(* IEC 61131-3 sources: eCockpitGit/test_project/src/%F%00 Library/%F%Common Functions/%F%Bits/%F%Bit Set Part Through, 8 files *)

(* ---- %POU%FU_bBitPartThrough.st ---- *)
//This function changed only the needed bits of a variable
// |**Version**|**Author**| **Date** |**Changes**
// | 1         | NSN      | 16-03-22 | Creation
FUNCTION FU_bBitPartThrough : BYTE
VAR_INPUT
	valueChange		:BYTE;		//Variable to change
	value			:BYTE;		//Value to change bits to
	amount			:BYTE;		//Amount of bits to change
	offset			:BYTE;		//Offset in variable to change bits at
END_VAR
(*%!%__DELIMITER__%!%*)
FU_bBitPartThrough		:=		(valueChange AND ROL(GConstants.binaryInvMaskByte[amount],offset)) OR SHL(value AND GConstants.binaryMaskByte[amount],offset);

(* ---- %POU%FU_diBitPartThrough.st ---- *)
//This function changed only the needed bits of a variable
// |**Version**|**Author**| **Date** |**Changes**
// | 1         | NSN      | 16-03-22 | Creation
FUNCTION FU_diBitPartThrough : DINT
VAR_INPUT
	valueChange		:DINT;		//Variable to change
	value			:DINT;		//Value to change bits to
	amount			:BYTE;		//Amount of bits to change
	offset			:BYTE;		//Offset in variable to change bits at
END_VAR
(*%!%__DELIMITER__%!%*)
FU_diBitPartThrough		:=		TO_DINT((TO_DWORD(valueChange) AND ROL(GConstants.binaryInvMaskDWord[amount],offset)) OR SHL(TO_DWORD(value) AND GConstants.binaryMaskDWord[amount],offset));

(* ---- %POU%FU_dwBitPartThrough.st ---- *)
//This function changed only the needed bits of a variable
// |**Version**|**Author**| **Date** |**Changes**
// | 1         | NSN      | 16-03-22 | Creation
FUNCTION FU_dwBitPartThrough : DWORD
VAR_INPUT
	valueChange		:DWORD;		//Variable to change
	value			:DWORD;		//Value to change bits to
	amount			:BYTE;		//Amount of bits to change
	offset			:BYTE;		//Offset in variable to change bits at
END_VAR
(*%!%__DELIMITER__%!%*)
FU_dwBitPartThrough		:=		(valueChange AND ROL(GConstants.binaryInvMaskDWord[amount],offset)) OR SHL(value AND GConstants.binaryMaskDWord[amount],offset);

(* ---- %POU%FU_iBitPartThrough.st ---- *)
//This function changed only the needed bits of a variable
// |**Version**|**Author**| **Date** |**Changes**
// | 1         | NSN      | 16-03-22 | Creation
FUNCTION FU_iBitPartThrough : INT
VAR_INPUT
	valueChange		:INT;		//Variable to change
	value			:INT;		//Value to change bits to
	amount			:BYTE;		//Amount of bits to change
	offset			:BYTE;		//Offset in variable to change bits at
END_VAR
(*%!%__DELIMITER__%!%*)
FU_iBitPartThrough		:=		TO_INT((TO_UINT(valueChange) AND ROL(TO_UINT(GConstants.binaryInvMaskInt[amount]),offset)) OR SHL(TO_UINT(value) AND TO_UINT(GConstants.binaryMaskInt[amount]),offset));

(* ---- %POU%FU_liBitPartThrough.st ---- *)
//This function changed only the needed bits of a variable
// |**Version**|**Author**| **Date** |**Changes**
// | 1         | NSN      | 16-03-22 | Creation
FUNCTION FU_liBitPartThrough : LINT
VAR_INPUT
	valueChange		:LINT;		//Variable to change
	value			:LINT;		//Value to change bits to
	amount			:BYTE;		//Amount of bits to change
	offset			:BYTE;		//Offset in variable to change bits at
END_VAR
(*%!%__DELIMITER__%!%*)
FU_liBitPartThrough		:=		TO_LINT((TO_LWORD(valueChange) AND ROL(GConstants.binaryInvMaskLWord[amount],offset)) OR SHL(TO_LWORD(value) AND GConstants.binaryMaskLWord[amount],offset));

(* ---- %POU%FU_lwBitPartThrough.st ---- *)
//This function changed only the needed bits of a variable
// |**Version**|**Author**| **Date** |**Changes**
// | 1         | NSN      | 16-03-22 | Creation
FUNCTION FU_lwBitPartThrough : LWORD
VAR_INPUT
	valueChange		:LWORD;		//Variable to change
	value			:LWORD;		//Value to change bits to
	amount			:BYTE;		//Amount of bits to change
	offset			:BYTE;		//Offset in variable to change bits at
END_VAR
(*%!%__DELIMITER__%!%*)
FU_lwBitPartThrough		:=		(valueChange AND ROL(GConstants.binaryInvMaskLWord[amount],offset)) OR SHL(value AND GConstants.binaryMaskLWord[amount],offset);

(* ---- %POU%FU_siBitPartThrough.st ---- *)
//This function changed only the needed bits of a variable
// |**Version**|**Author**| **Date** |**Changes**
// | 1         | NSN      | 16-03-22 | Creation
FUNCTION FU_siBitPartThrough : SINT
VAR_INPUT
	valueChange		:SINT;		//Variable to change
	value			:SINT;		//Value to change bits to
	amount			:BYTE;		//Amount of bits to change
	offset			:BYTE;		//Offset in variable to change bits at
END_VAR
(*%!%__DELIMITER__%!%*)
FU_siBitPartThrough		:=		TO_SINT((TO_USINT(valueChange) AND ROL(TO_USINT(GConstants.binaryInvMaskSint[amount]),offset)) OR SHL(TO_USINT(value) AND TO_USINT(GConstants.binaryMaskSint[amount]),offset));

(* ---- %POU%FU_wBitPartThrough.st ---- *)
//This function changed only the needed bits of a variable
// |**Version**|**Author**| **Date** |**Changes**
// | 1         | NSN      | 16-03-22 | Creation
FUNCTION FU_wBitPartThrough : WORD
VAR_INPUT
	valueChange		:WORD;		//Variable to change
	value			:WORD;		//Value to change bits to
	amount			:BYTE;		//Amount of bits to change
	offset			:BYTE;		//Offset in variable to change bits at
END_VAR
(*%!%__DELIMITER__%!%*)
FU_wBitPartThrough		:=		(valueChange AND ROL(GConstants.binaryInvMaskWord[amount],offset)) OR SHL(value AND GConstants.binaryMaskWord[amount],offset);
